(* PLC project Unnamed, Unknown Unnamed 1 *)
(* stored: creationDateTime 2025-11-05T10:53:43, modificationDateTime 2025-11-05T11:11:27 *)

PROGRAM main
  VAR
    Trigger : BOOL := False;
    F_Triggered : BOOL := False;
    EStop_Ok : BOOL := True;
    Fault_Timeout : BOOL := False;
    Safe : BOOL := False;
    Running : BOOL := True;
    InPosition : BOOL := False;
    Command : BOOL := False;
    FaultReset : BOOL := False;
    Sensor : BOOL := False;
    F_Triggered8 : BOOL := False;
    T_Fault : TON;
  END_VAR

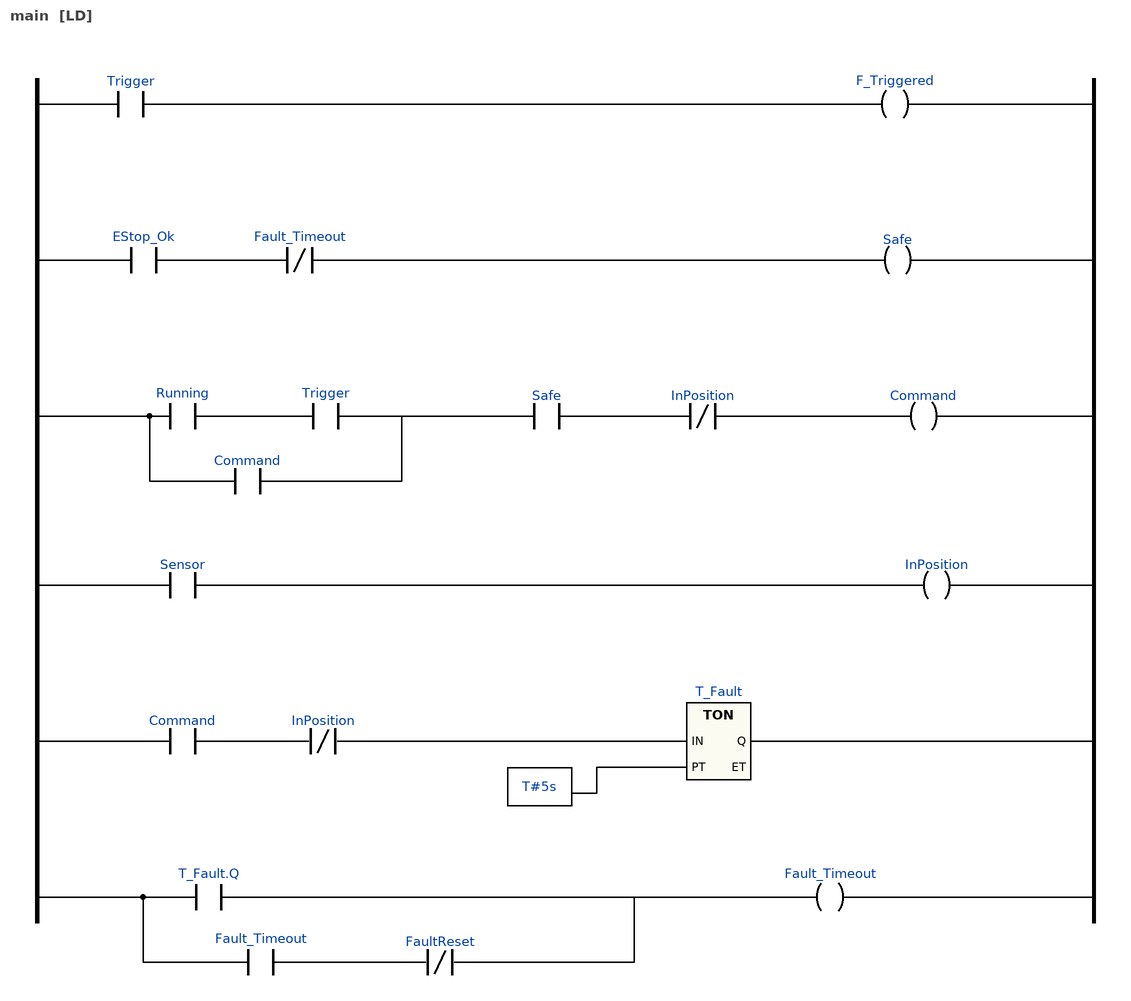
(* LD diagram, written out as Structured Text *)
F_Triggered := Trigger;
Safe := EStop_Ok AND NOT Fault_Timeout;
Command := (Running AND Trigger OR Command) AND Safe AND NOT InPosition;
InPosition := Sensor;
Fault_Timeout := T_Fault.Q OR Fault_Timeout AND NOT FaultReset;
T_Fault(IN := Command AND NOT InPosition, PT := T#5s);
END_PROGRAM

CONFIGURATION Config0
  RESOURCE Res0 ON PLC
    TASK task0(INTERVAL := T#20ms, PRIORITY := 0);
    PROGRAM instance0 WITH task0 : main;
  END_RESOURCE
END_CONFIGURATION
